{attribute 'GeneratedUsingTerminal: KL6224-0002'}
{attribute addProperty BoxType "KL6224-0002"}
{attribute addProperty Description ""}
{attribute addProperty Physics ""}
{attribute addProperty Id "Channel_1AT %Q*Channel_A04AC4BD0"}
{attribute addProperty CRC "3306888368"}
{attribute addProperty Size "0"}
TYPE KL_C51B1CB0 :
STRUCT
	{attribute addProperty Name "Channel_1"}
	Channel_1 : Channel_A04AC4BD;
END_STRUCT
END_TYPE

(* stored: Version 1.2.0.0, ProductVersion 3.1.4024.11
   DUT KL_C51B1CB0: Id {3232cf7a-f0a4-411a-b2ae-6e712e13f50a} *)
